FUNCTION_BLOCK PUBLIC FB_Conveyor

VAR_IN_OUT
	HardwareInputArray : ARRAY [*] OF BOOL;		// For Actuators
END_VAR

VAR
	Configuration 	: ST_ConveyorConfiguration;
	Controls		: ST_ConveyorControls;
	Status			: ST_ConveyorStatus;
	
	InitDone 		: BOOL := FALSE;
	
	State			: DINT := E_ConveyorStates.Stopped;
	Running			: BOOL := FALSE; // Controls conveyor running, Initialized false to ensure conveyors are off on startup
END_VAR

IF NOT InitDone THEN
	M_Init();
	InitDone:= TRUE;
ELSE
	M_Cyclic();
	M_StateMachine();
END_IF

METHOD PRIVATE M_Cyclic : BOOL
Configuration.OutputArrayPosition := Configuration.HardwareOutput - 32768;
HardwareInputArray[Configuration.OutputArrayPosition] := Running;
Status.isRunning := Running;
END_METHOD

METHOD PRIVATE M_Init : BOOL
VAR
END_VAR
END_METHOD

METHOD PUBLIC M_Reset : BOOL
VAR_INPUT
END_VAR
END_METHOD

METHOD PRIVATE M_StateMachine : BOOL
CASE State OF
	E_ConveyorStates.Stopped: 
		IF Controls.RequestRun THEN
			State := E_ConveyorStates.RunRequest;
			Controls.RequestRun := FALSE;
		END_IF
		
	E_ConveyorStates.RunRequest:
		Running := TRUE;
		State := E_ConveyorStates.Running;
		
	E_ConveyorStates.Running:
		IF Controls.RequestStop THEN
			State := E_ConveyorStates.StopRequest;
			Controls.RequestStop := FALSE;
		END_IF
		
	E_ConveyorStates.StopRequest:
		Running := FALSE;
		State := E_ConveyorStates.Stopped;
		
END_CASE
END_METHOD

PROPERTY P_Configuration : REFERENCE TO ST_ConveyorConfiguration
GET // PUBLIC
P_Configuration REF= Configuration;
END_GET
END_PROPERTY

PROPERTY PUBLIC P_Controls : REFERENCE TO ST_ConveyorControls
GET // PUBLIC
P_Controls REF= Controls;
END_GET
END_PROPERTY

PROPERTY P_Status : REFERENCE TO ST_ConveyorStatus
GET
P_Status REF= Status;
END_GET
END_PROPERTY

END_FUNCTION_BLOCK

(* stored: Version 1.1.0.1, ProductVersion 3.1.4024.12
   POU FB_Conveyor: Id {795138f7-32e1-4f4d-be5d-521d4edc8b59}, SpecialFunc None
   Method M_Cyclic: Id {9c7b7699-b261-439a-af2c-8ff428580a73}
   Method M_Init: Id {f38c6018-898d-4472-8b72-b1c3b7ede863}
   Method M_Reset: Id {0f31457f-3c8a-4ef8-a73a-775dcd954453}
   Method M_StateMachine: Id {f557a3e8-a4dc-4150-bcb7-ea5da06edf1f}
   Property P_Configuration: Id {cdfbb0d5-3782-4885-803d-95c81bda4d95}
   Get Get: Id {9a053f5a-5c04-4402-a515-60b8aa436ba6}
   Property P_Controls: Id {16d97001-52f1-42da-9f4c-7af3f68852d8}
   Get Get: Id {496a1c07-8e8e-40b2-bdae-0f4961766996}
   Property P_Status: Id {4a132a40-2714-4c36-8475-81001e1683b1}
   Get Get: Id {376e1ab0-4ce3-411e-818b-82c500ce5092} *)
